ABB RobotStudio station: Task1_welding.rspag

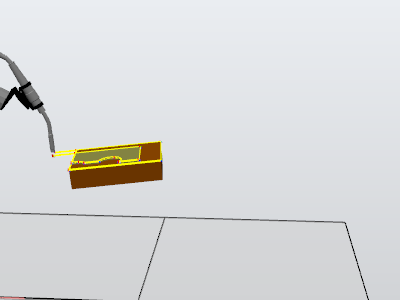
--- station ---
Station Task1_welding (saved by RobotStudio 24.3.10958.1)
Controller IRB_1520ID_4kg_1.50m
  mechanical unit ROB_1: IRB1520ID_4_150__02, 6 joints, base frame (0, 0, 0) mm
Layout (positions relative to the parent item):
  - IRB1520ID_4_150__02 [mechanism, from %ABB.RobotStudio.Models.IRB1520ID%\IRB1520ID_4_150_G_02.rslib] at (0, 0, 0) mm; joint values [1.0873, -1.1398, 1.0927, -0.9268, 1.0857, 1.1884] (rad or m)
  - AW_Gun_PSF_25 [mechanism, from %ABB.RobotStudio.Models.ArcWelding%\AW_Gun_PSF_25.rslib] at (327.45, 319.27, 831.55) mm, rotated rx -180 ry 59.43 rz -172.96 deg
  - Curve_thing [part, from Training Objects\Curve_Thing.rslib] at (696.55, 149.94, 458.64) mm, rotated rx 0 ry -5.23 rz 7.04 deg
Attachment: AW_Gun_PSF_25 is attached to IRB1520ID_4_150__02 / Link6

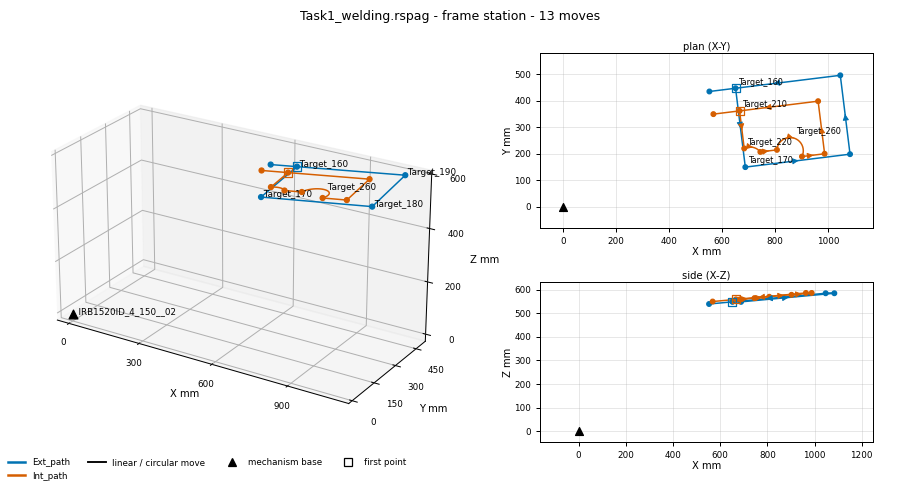
[picture p0: tool path of Task1_welding.rspag in frame station, 13 of 15 moves have a stored position in this frame; points joined in program order, loops and branches not executed]
--- Backups/IRB_1520ID_4kg_1.50m/RAPID/TASK1/PROGMOD/CalibData.mod ---
MODULE CalibData
	PERS tooldata AW_Gun:=[TRUE,[[119.5,0,352],[0.890213743,0,0.455543074,0]],[1,[0,0,100],[1,0,0,0],0,0,0]];
	TASK PERS wobjdata myPalletWO:=[FALSE,TRUE,"",[[688.418839009,148.925896983,548.269503166],[0.74843401,0.03415564,-0.030194721,-0.66164054]],[[0,0,0],[1,0,0,0]]];
    TASK PERS wobjdata Workobject_1:=[FALSE,TRUE,"",[[1083.749,197.778,584.702],[0.04550354,-0.061367918,0.997073499,0.002800654]],[[0,0,0],[1,0,0,0]]];
ENDMODULE

--- Backups/IRB_1520ID_4kg_1.50m/RAPID/TASK1/PROGMOD/Module1.mod ---
MODULE Module1


    CONST robtarget Target_160:=[[400.002823158,299.996341704,-0.001267742],[1,0,0,0],[0,0,0,0],[9E+09,9E+09,9E+09,9E+09,9E+09,9E+09]];
    CONST robtarget Target_170:=[[400.000217389,-0.003658284,-0.00102963],[1,0,0,0],[0,0,0,0],[9E+09,9E+09,9E+09,9E+09,9E+09,9E+09]];
    CONST robtarget Target_180:=[[0.000217404,-0.000183925,-0.000514684],[1,0,0,0],[0,0,0,0],[9E+09,9E+09,9E+09,9E+09,9E+09,9E+09]];
    CONST robtarget Target_190:=[[0.002823174,299.999816064,-0.000752796],[1,0,0,0],[0,0,0,0],[9E+09,9E+09,9E+09,9E+09,9E+09,9E+09]];
    CONST robtarget Target_200:=[[400.002823158,299.996341704,-0.001267742],[1,0,0,0],[0,0,0,0],[9E+09,9E+09,9E+09,9E+09,9E+09,9E+09]];
    CONST robtarget Target_210:=[[394.55428828,213.322552964,-10.001191935],[1,0,0,0],[0,0,0,0],[9E+09,9E+09,9E+09,9E+09,9E+09,9E+09]];
    CONST robtarget Target_220:=[[394.553047294,70.449008728,-10.001078535],[1,0,0,0],[0,0,0,0],[9E+09,9E+09,9E+09,9E+09,9E+09,9E+09]];
    CONST robtarget Target_230:=[[361.411159423,70.599394567,-10.001035989],[1,0,0,0],[0,0,0,0],[9E+09,9E+09,9E+09,9E+09,9E+09,9E+09]];
    CONST robtarget Target_240:=[[335.455881543,49.990394162,-10.000986218],[1,0,0,0],[0,0,0,0],[9E+09,9E+09,9E+09,9E+09,9E+09,9E+09]];
    CONST robtarget Target_250:=[[272.035683499,49.990945024,-10.000904572],[1,0,0,0],[0,0,0,0],[9E+09,9E+09,9E+09,9E+09,9E+09,9E+09]];
    CONST robtarget Target_260:=[[204.241372168,86.97886701,-10.000846653],[1,0,0,0],[0,0,0,0],[9E+09,9E+09,9E+09,9E+09,9E+09,9E+09]];
    CONST robtarget Target_270:=[[181.020785538,13.324407687,-10.000758301],[1,0,0,0],[0,0,0,0],[9E+09,9E+09,9E+09,9E+09,9E+09,9E+09]];
    CONST robtarget Target_280:=[[94.552551112,13.325158742,-10.000646984],[1,0,0,0],[0,0,0,0],[9E+09,9E+09,9E+09,9E+09,9E+09,9E+09]];
    CONST robtarget Target_290:=[[94.554288291,213.325158734,-10.000805725],[1,0,0,0],[0,0,0,0],[9E+09,9E+09,9E+09,9E+09,9E+09,9E+09]];
    CONST robtarget Target_300:=[[394.55428828,213.322552964,-10.001191935],[1,0,0,0],[0,0,0,0],[9E+09,9E+09,9E+09,9E+09,9E+09,9E+09]];


    PROC main()
        WHILE TRUE DO
           Ext_path;
           Int_path;
           WaitTime 3;
        ENDWHILE
    ENDPROC

    PROC Ext_path()
        VAR robtarget top_160;
        top_160:=Offs(Target_160,0,0,-100);

        MoveJ top_160,v500,z100,AW_Gun\WObj:=Workobject_1;
        MoveL Target_160,v100,fine,AW_Gun\WObj:=Workobject_1;
        MoveL Target_170,v300,fine,AW_Gun\WObj:=Workobject_1;
        MoveL Target_180,v300,fine,AW_Gun\WObj:=Workobject_1;
        MoveL Target_190,v300,fine,AW_Gun\WObj:=Workobject_1;
        MoveL Offs(Target_200,100,0,0),v300,z100,AW_Gun\WObj:=Workobject_1;
    ENDPROC

    PROC Int_path()
        VAR robtarget top_210;
        top_210:=Offs(Target_210,0,0,-100);

        MoveJ top_210,v500,z100,AW_Gun\WObj:=Workobject_1;
        MoveL Target_210,v100,fine,AW_Gun\WObj:=Workobject_1;
        MoveL Target_220,v300,fine,AW_Gun\WObj:=Workobject_1;
        MoveC Target_230,Target_240,v300,fine,AW_Gun\WObj:=Workobject_1;
        MoveL Target_250,v300,fine,AW_Gun\WObj:=Workobject_1;
        MoveC Target_260,Target_270,v300,fine,AW_Gun\WObj:=Workobject_1;
        MoveL Target_280,v300,fine,AW_Gun\WObj:=Workobject_1;
        MoveL Target_290,v300,fine,AW_Gun\WObj:=Workobject_1;
        MoveL Offs(Target_300,100,0,0),v300,fine,AW_Gun\WObj:=Workobject_1;
    ENDPROC

ENDMODULE

--- Backups/IRB_1520ID_4kg_1.50m/RAPID/TASK1/SYSMOD/LINKEDM.sys ---
%%%
  VERSION:1
  LANGUAGE:ENGLISH
%%%

MODULE LINKEDM (SYSMODULE)

! FOLLOWER
!     Name of electronically linked follower axis used by operator at teach pendent.
      PERS string l_f_axis_name{5}       :=  ["",  "", "", "", ""];

!     Name of the mechanical unit for follower axis.
      PERS string l_f_mecunt_n{5}  :=  ["", "", "", "", ""];

!     Linked follower axis number in the mechanical unit (first axis in mech. unit is number 1).
      PERS num l_f_axis_no{5}      :=  [0,          0,   0,  0,  0];

! MASTER
!     Name of the mechanical unit for linked master axis.
      PERS string l_m_mecunt_n{5} :=  ["", "", "", "", ""];

!     Linked master axis number in the mechanical unit (first axis in mech. unit is number 1).
!     See axis number table in documentation for different master mechanical units.
      PERS num l_m_axis_no{5}     :=  [0,  0,  0,  0,  0];

! POSITION OFFSET
!     The increase of the allowed offset position between the master and follower
!     positions, used when starting AUTO mode. As soon as the offset is decreased
!     the old configurated parameter is used.
!     Example: 3 => the configurated value of allowed offset is increased 3 times.
      PERS num offset_ratio{5}       :=  [10,  10,   10,  10,  10];

! SPEED RATIO
!     Speed_ratio used in AUTO and JOG modes [ very_slow   slow    normal    fast]
!     Value 1 = max allowed manual speed.
      CONST num speed_ratio {20}      := [0.01, 0.01, 0.01, 0.01, 0.01,
                                          0.05, 0.05, 0.05, 0.05, 0.05,
                                          0.20, 0.20, 0.20, 0.20, 0.20,
                                          1.00, 1.00, 1.00, 1.00, 1.00];

! STEP SIZE
!     Displacement position used in JOG mode for each activation of positive or
!     negative movement.                  [very_short    short   normal   long]
!     Unit degees or meter.
      CONST num displacement {20}     := [0.001, 0.001, 0.001, 0.001, 0.001,
                                          0.005, 0.005, 0.005, 0.005, 0.005,
                                          0.020, 0.020, 0.020, 0.020, 0.020,
                                          0.100, 0.100, 0.100, 0.100, 0.100];


!-------------------------------------------------------------
 PROC Linked_m ()
      Linked_m_exe ;
 ENDPROC
ENDMODULE

--- Backups/IRB_1520ID_4kg_1.50m/SYSPAR/EIO.cfg ---
EIO:CFG_1.0:6:1::
#
EIO_SIGNAL:

      -Name "MyDO1" -SignalType "DO"

      -Name "MyDO2" -SignalType "DO"
